// TwinCAT 3 PLC project TcCylinder
// Title: TcCylinder
// Company: TcNexa
// Author: ATI Software Engineering
// ProjectVersion: 2.2.0
// ProgramVersion: 3.1.4026.20
// libraries:
//   Tc2_Standard, * (Beckhoff Automation GmbH)
//   Tc2_System, * (Beckhoff Automation GmbH)
//   Tc3_Module, * (Beckhoff Automation GmbH)
//   TcDeviceBase, * (TcNexa)
//   TcProcess, * (TcNexa)
//   TcUnit, * (www.tcunit.org)
//   TcUtilities, * (TcNexa)
// project tree:
//   Cylinder/DUTs/ ST_CylinderConfig.TcDUT, ST_CylinderInfo.TcDUT
//   Cylinder/ITFs/ I_Cylinder.TcIO
//   Cylinder/POUs/ FB_Cylinder.TcPOU, FB_LiftCylinderBosch.TcPOU, FB_CylinderNexaHmi.TcPOU, FB_LiftCylinderNexaHmi_Bosch.TcPOU
//   / PlcTask.TcTTO
//   Tests/ FB_Cylinder_Test.TcPOU, PRG_TEST.TcPOU
//   Version/ Global_Version.TcGVL
// real-time tasks:
//   TASK PlcTask: cycle T#10ms, priority 20, ADS port 350

CONFIGURATION TcCylinder
    RESOURCE PLC ON TwinCAT3
        TASK PlcTask(INTERVAL := T#10ms, PRIORITY := 20);
        PROGRAM PRG_TEST WITH PlcTask : PRG_TEST;
    END_RESOURCE
END_CONFIGURATION

// ---- Cylinder/DUTs/ST_CylinderConfig.TcDUT
TYPE INTERNAL ST_CylinderConfig :
STRUCT
	delayTimeAfterReachedHP		: TIME;
	delayTimeAfterReachedWP		: TIME;
	movementTimeout				: TIME:= T#5S;
	monitorSensorsOverlap		: BOOL:= TRUE;
	sensorsOverlapTimeout		: TIME:= T#100MS;
END_STRUCT
END_TYPE

// ---- Cylinder/DUTs/ST_CylinderInfo.TcDUT
TYPE INTERNAL ST_CylinderInfo :
STRUCT
	sensorHP			: BOOL;
	sensorWP			: BOOL;
END_STRUCT
END_TYPE

// ---- Version/Global_Version.TcGVL
{attribute 'TcGenerated'}
{attribute 'no-analysis'}
{attribute 'linkalways'}
// This function has been automatically generated from the project information.
VAR_GLOBAL CONSTANT
	{attribute 'const_non_replaced'}
	stLibVersion_TcCylinder : ST_LibVersion := (iMajor := 2, iMinor := 2, iBuild := 0, iRevision := 0, nFlags := 0, sVersion := '2.2.0');
END_VAR

// ---- Cylinder/ITFs/I_Cylinder.TcIO
INTERFACE I_Cylinder

METHOD fill
VAR_INPUT
END_VAR
END_METHOD

PROPERTY PUBLIC inHP : BOOL
GET
END_GET
END_PROPERTY

PROPERTY PUBLIC inWP : BOOL
GET
END_GET
END_PROPERTY

METHOD PUBLIC moveToHP
VAR_INPUT
	Response		: REFERENCE TO TcNexa_Components_TcProcess.FB_MethodResponse;
END_VAR
END_METHOD

METHOD PUBLIC moveToWP
VAR_INPUT
	Response		: REFERENCE TO TcNexa_Components_TcProcess.FB_MethodResponse;
END_VAR
END_METHOD

METHOD PUBLIC off
VAR_INPUT
END_VAR
END_METHOD

END_INTERFACE

// ---- Tests/PRG_TEST.TcPOU
PROGRAM PRG_TEST
VAR
	_test : FB_Cylinder_Test;
END_VAR

TcUnit.RUN();

END_PROGRAM

// ---- Tests/FB_Cylinder_Test.TcPOU
FUNCTION_BLOCK FB_Cylinder_Test EXTENDS TcUnit.FB_TestSuite
VAR
END_VAR

testMoveToHP_BothSensorActive_Error();
testMoveToHP_MovementInterlocked_Error();
testMoveToHP_SensorNotReached_Timeout();
testMoveToHP_SensorNotUsed_Ok();
testMoveToHP_SensorReached_Ok();

METHOD PROTECTED testMoveToHP_BothSensorActive_Error
VAR_INST
	_testTimeout		: Tc2_Standard.TON;
	_Cylinder 			: FB_Cylinder	(name		:= 'Cylinder',
										tag			:= 'C1',
										sensorTagHP	:= 'B1',
										sensorTagWP	:= 'B2');
	_Response			: TcNexa_Components_TcProcess.FB_MethodResponse;
	_timerDelay			: Tc2_Standard.TON;
END_VAR
IF TcUnit.TEST_ORDERED(TestName:= 'TestMoveToHP_BothSensorActive_Error') THEN
	// Timeout if the movement is not executed right
	_testTimeout(IN:= TRUE, PT:= T#10S);
	_timerDelay(IN:= TRUE, PT:= T#1S);
	// Cylinder call
	_Cylinder.Config.delayTimeAfterReachedHP:= T#1S;	
	_Cylinder.FB_main();
	_Cylinder.moveToHP(Response:= _Response);
	TcUnit.WRITE_PROTECTED_BOOL(Ptr:= ADR(_Cylinder.sensorHP), Value:= _timerDelay.Q);
	TcUnit.WRITE_PROTECTED_BOOL(Ptr:= ADR(_Cylinder.sensorWP), Value:= TRUE);
	// Wait result
	IF _testTimeout.Q OR _Cylinder.inHP OR NOT _Response.busy THEN
		AssertFalse(
			Condition	:= _Cylinder.inHP,
			Message		:= 'inHP not FALSE');
		AssertFalse(
			Condition	:= _Cylinder.inWP,
			Message		:= 'inWP not FALSE');
		AssertFalse(
			Condition	:= _Response.busy,
			Message		:= 'busy not FALSE');
		AssertTrue(
			Condition	:= _Response.error,
			Message		:= 'error not TRUE');
			
		TcUnit.TEST_FINISHED();
	END_IF
END_IF
END_METHOD

METHOD PROTECTED testMoveToHP_MovementInterlocked_Error
VAR_INST
	_testTimeout		: Tc2_Standard.TON;
	_Cylinder 			: FB_Cylinder	(name		:= 'Cylinder',
										tag			:= 'C1',
										sensorTagHP	:= 'B1',
										sensorTagWP	:= 'B2');
	_Response			: TcNexa_Components_TcProcess.FB_MethodResponse;
	_timerDelay			: Tc2_Standard.TON;
END_VAR
IF TcUnit.TEST_ORDERED(TestName:= 'testMoveToHP_MovementInterlocked_Error') THEN
	// Timeout if the movement is not executed right
	_testTimeout(IN:= TRUE, PT:= T#10S);
	_timerDelay(IN:= TRUE, PT:= T#1S);
	// Cylinder call
	_Cylinder.addInterlockHP(condition:= TRUE, message:= '');
	_Cylinder.FB_main();
	_Cylinder.moveToHP(Response:= _Response);
	TcUnit.WRITE_PROTECTED_BOOL(Ptr:= ADR(_Cylinder.sensorHP), Value:= _timerDelay.Q);
	// Wait result
	IF _testTimeout.Q OR _Cylinder.inHP OR NOT _Response.busy THEN
		AssertFalse(
			Condition	:= _Cylinder.inHP,
			Message		:= 'inHP not FALSE');
		AssertFalse(
			Condition	:= _Cylinder.inWP,
			Message		:= 'inWP not FALSE');
		AssertFalse(
			Condition	:= _Response.busy,
			Message		:= 'busy not FALSE');
		AssertTrue(
			Condition	:= _Response.error,
			Message		:= 'error not TRUE');
			
		TcUnit.TEST_FINISHED();
	END_IF
END_IF
END_METHOD

METHOD PROTECTED testMoveToHP_SensorNotReached_Timeout
VAR_INST
	_testTimeout		: Tc2_Standard.TON;
	_Cylinder 			: FB_Cylinder	(name		:= 'Cylinder',
										tag			:= 'C1',
										sensorTagHP	:= 'B1',
										sensorTagWP	:= 'B2');
	_Response			: TcNexa_Components_TcProcess.FB_MethodResponse;
END_VAR
IF TcUnit.TEST_ORDERED(TestName:= 'TestMoveToHP_SensorNotReached_Timeout') THEN
	// Timeout if the movement is not executed right
	_testTimeout(IN:= TRUE, PT:= T#10S);
	// Cylinder call
	_Cylinder.FB_main();
	_Cylinder.moveToHP(Response:= _Response);
	// Wait result
	IF _testTimeout.Q OR _Cylinder.inHP OR NOT _Response.busy THEN
		AssertFalse(
			Condition	:= _Cylinder.inHP,
			Message		:= 'inHP not FALSE');
		AssertFalse(
			Condition	:= _Cylinder.inWP,
			Message		:= 'inWP not FALSE');
		AssertFalse(
			Condition	:= _Response.busy,
			Message		:= 'busy not FALSE');
		AssertTrue(
			Condition	:= _Response.error,
			Message		:= 'error not TRUE');
			
		TcUnit.TEST_FINISHED();
	END_IF
END_IF
END_METHOD

METHOD PROTECTED testMoveToHP_SensorNotUsed_Ok
VAR_INST
	_testTimeout		: Tc2_Standard.TON;
	_Cylinder 			: FB_Cylinder	(name		:= 'Cylinder',
										tag			:= 'C1',
										sensorTagHP	:= '',
										sensorTagWP	:= 'B2');
	_Response			: TcNexa_Components_TcProcess.FB_MethodResponse;
END_VAR
IF TcUnit.TEST_ORDERED(TestName:= 'testMoveToHP_SensorNotUsed_Ok') THEN
	// Timeout if the movement is not executed right
	_testTimeout(IN:= TRUE, PT:= T#10S);
	// Cylinder call
	_Cylinder.Config.delayTimeAfterReachedHP:= T#1S;
	_Cylinder.FB_main();
	_Cylinder.moveToHP(Response:= _Response);
	// Wait result
	IF _testTimeout.Q OR _Cylinder.inHP OR NOT _Response.busy THEN
		AssertTrue(
			Condition	:= _Cylinder.inHP,
			Message		:= 'inHP not TRUE');
		AssertFalse(
			Condition	:= _Cylinder.inWP,
			Message		:= 'inWP not FALSE');
		AssertFalse(
			Condition	:= _Response.busy,
			Message		:= 'busy not FALSE');
		AssertFalse(
			Condition	:= _Response.error,
			Message		:= 'error not FALSE');
			
		TcUnit.TEST_FINISHED();
	END_IF
END_IF
END_METHOD

METHOD PROTECTED testMoveToHP_SensorReached_Ok
VAR_INST
	_testTimeout		: Tc2_Standard.TON;
	_Cylinder 			: FB_Cylinder	(name		:= 'Cylinder',
										tag			:= 'C1',
										sensorTagHP	:= 'B1',
										sensorTagWP	:= 'B2');
	_Response			: TcNexa_Components_TcProcess.FB_MethodResponse;
	_timerDelay			: Tc2_Standard.TON;
END_VAR
IF TcUnit.TEST_ORDERED(TestName:= 'TestMoveToHP_SensorReached_Ok') THEN
	// Timeout if the movement is not executed right
	_testTimeout(IN:= TRUE, PT:= T#10S);
	_timerDelay(IN:= TRUE, PT:= T#1S);
	// Cylinder call
	_Cylinder.Config.delayTimeAfterReachedHP:= T#1S;	
	_Cylinder.FB_main();
	_Cylinder.moveToHP(Response:= _Response);
	TcUnit.WRITE_PROTECTED_BOOL(Ptr:= ADR(_Cylinder.sensorHP), Value:= _timerDelay.Q);
	// Wait result
	IF _testTimeout.Q OR _Cylinder.inHP OR NOT _Response.busy THEN
		AssertTrue(
			Condition	:= _Cylinder.inHP,
			Message		:= 'inHP not TRUE');
		AssertFalse(
			Condition	:= _Cylinder.inWP,
			Message		:= 'inWP not FALSE');
		AssertFalse(
			Condition	:= _Response.busy,
			Message		:= 'busy not FALSE');
		AssertFalse(
			Condition	:= _Response.error,
			Message		:= 'error not FALSE');
		AssertEquals_TIME(
			Expected	:= _timerDelay.ET + _Cylinder.Config.delayTimeAfterReachedHP + T#10MS,
			Actual		:= _testTimeout.ET,
			Message		:= 'delayTimeAfterReachedHP missmatch');
			
		TcUnit.TEST_FINISHED();
	END_IF
END_IF
END_METHOD

END_FUNCTION_BLOCK

// ---- Cylinder/POUs/FB_Cylinder.TcPOU
FUNCTION_BLOCK FB_Cylinder EXTENDS TcNexa_Devices_TcDeviceBase.FB_DeviceBase IMPLEMENTS I_Cylinder
VAR
(*----------------------------------------------------------------------------------------------*)
	sensorHP		AT %I*		: BOOL;
	sensorWP		AT %I*		: BOOL;
	valveHP			AT %Q*		: BOOL;
	valveWP			AT %Q*		: BOOL;
(*----------------------------------------------------------------------------------------------*)
	_Config						: ST_CylinderConfig;
	_Info						: ST_CylinderInfo;
	_inHP						: BOOL;
	_inWP						: BOOL;
	_newStateInterlockHP		: BOOL;
	_newStateInterlockMsgHP		: STRING(255);
	_interlockHP				: BOOL;
	_interlockMessageHP			: STRING(255);
	_newStateInterlockWP		: BOOL;
	_newStateInterlockMsgWP		: STRING(255);
	_interlockWP				: BOOL;
	_interlockMessageWP			: STRING(255);
	_sensorTagHP				: STRING;
	_sensorTagWP				: STRING;
	_notUsedSensorHP			: BOOL;
	_notUsedSensorWP			: BOOL;
	_timerTimeout				: Tc2_Standard.TON;
	_timerSensorsOverlap		: Tc2_Standard.TON;
	_timerInHP					: Tc2_Standard.TON;
	_timerInWP					: Tc2_Standard.TON;
(*----------------------------------------------------------------------------------------------*)
END_VAR

METHOD INTERNAL _getErrorMsgPositionNotReached : STRING(255)
VAR_INPUT
	sensor		: STRING;
END_VAR
_getErrorMsgPositionNotReached:= 'Position not reached';
IF (sensor <> '') THEN
	_getErrorMsgPositionNotReached:= Tc2_Standard.CONCAT(STR1:= _getErrorMsgPositionNotReached, STR2:= ' (');
	_getErrorMsgPositionNotReached:= Tc2_Standard.CONCAT(STR1:= _getErrorMsgPositionNotReached, STR2:= sensor);
	_getErrorMsgPositionNotReached:= Tc2_Standard.CONCAT(STR1:= _getErrorMsgPositionNotReached, STR2:= ')');
END_IF
END_METHOD

METHOD INTERNAL _getMsgInterlocked : STRING(255)
VAR_INPUT
END_VAR
_getMsgInterlocked:= Tc2_Standard.CONCAT(STR1:= _nameTag, STR2:= ' interlocked during ');
_getMsgInterlocked:= Tc2_Standard.CONCAT(STR1:= _getMsgInterlocked, STR2:= _calledMethod);
END_METHOD

METHOD INTERNAL _handleInterlocks
VAR_INPUT
END_VAR
(*----------------------------------------------------------------------------------------------*)
_interlockHP:= _newStateInterlockHP;
_interlockMessageHP:= _newStateInterlockMsgHP;
_newStateInterlockHP:= FALSE;
_newStateInterlockMsgHP:= '';
(*----------------------------------------------------------------------------------------------*)
_interlockWP:= _newStateInterlockWP;
_interlockMessageWP:= _newStateInterlockMsgWP;
_newStateInterlockWP:= FALSE;
_newStateInterlockMsgWP:= '';
(*----------------------------------------------------------------------------------------------*)
END_METHOD

METHOD INTERNAL _handlePositionStatus
VAR_INPUT
END_VAR
(*----------------------------------------------------------------------------------------------*)
_timerInHP(
	IN	:= valveHP AND (_notUsedSensorHP OR sensorHP) AND (NOT sensorWP OR NOT _Config.monitorSensorsOverlap),
	PT	:= _Config.delayTimeAfterReachedHP,
	Q	=> _inHP);
(*----------------------------------------------------------------------------------------------*)
_timerInWP(
	IN	:= valveWP AND (_notUsedSensorWP OR sensorWP) AND (NOT sensorHP OR NOT _Config.monitorSensorsOverlap),
	PT	:= _Config.delayTimeAfterReachedWP,
	Q	=> _inWP);
(*----------------------------------------------------------------------------------------------*)
_timerTimeout(
	IN:= (_calledMethod <> ''),
	PT:= _Config.movementTimeout);
(*----------------------------------------------------------------------------------------------*)
_timerSensorsOverlap(
	IN:= _Config.monitorSensorsOverlap AND sensorHP AND sensorWP,
	PT:= _Config.sensorsOverlapTimeout);
(*----------------------------------------------------------------------------------------------*)
END_METHOD

METHOD PROTECTED _methodHeader : ST_MethodState
VAR_INPUT
	methodName		: Tc2_System.T_MaxString;
END_VAR
IF (_calledMethod = '') THEN
	_timerTimeout(IN:= FALSE);
	_timerSensorsOverlap(IN:= FALSE);
	_calledMethod:= methodName;
	_Step.init();
	_methodTimeout(IN:= FALSE);
	_methodHeader.init:= TRUE;
	_methodHeader.execute:= TRUE;
	_executeMethod:= TRUE;
	_InternalResponse.setBusy(message:= methodName);
ELSIF (_calledMethod = methodName) THEN
	_executeMethod:= TRUE;
	_tmpText:= _getBusyMessage(message:= 'in progress');
	_InternalResponse.setBusy(message:= _tmpText);
	_methodHeader.execute:= TRUE;
ELSE
	_tmpText:= _getBusyMessage(message:= 'in progress');
	_InternalResponse.setBusy(message:= _tmpText);
END_IF
END_METHOD

METHOD PROTECTED _onInit
VAR_INST
	_isInit				: BOOL;
END_VAR
(*----------------------------------------------------------------------------------------------*)
IF _isInit THEN RETURN; END_IF
(*----------------------------------------------------------------------------------------------*)
IF (_sensorTagHP = '') THEN
	_notUsedSensorHP:= TRUE;
END_IF
(*----------------------------------------------------------------------------------------------*)
IF (_sensorTagWP = '') THEN
	_notUsedSensorWP:= TRUE;
END_IF
(*----------------------------------------------------------------------------------------------*)
_isInit:= TRUE;
(*----------------------------------------------------------------------------------------------*)
END_METHOD

METHOD INTERNAL _updateInfo
VAR_INPUT
END_VAR
_Info.sensorHP:= sensorHP;
_Info.sensorWP:= sensorWP;
END_METHOD

METHOD addInterlockHP
VAR_INPUT
	condition		: BOOL;
	message			: STRING(255);
END_VAR
IF condition THEN
	_newStateInterlockHP:= TRUE;
	_newStateInterlockMsgHP:= message;
END_IF
END_METHOD

METHOD addInterlockWP
VAR_INPUT
	condition		: BOOL;
	message			: STRING(255);
END_VAR
IF condition THEN
	_newStateInterlockWP:= TRUE;
	_newStateInterlockMsgWP:= message;
END_IF
END_METHOD

PROPERTY Config : REFERENCE TO ST_CylinderConfig
GET
Config REF= _Config;
END_GET
END_PROPERTY

METHOD FB_init : BOOL
VAR_INPUT
	bInitRetains 	: BOOL; 	// if TRUE, the retain variables are initialized (warm start / cold start)
	bInCopyCode 	: BOOL;  	// if TRUE, the instance afterwards gets moved into the copy code (online change)
	name			: STRING;	// identifier for HMI display and logging, example Clipping cylinder
	tag				: STRING;	// el. schematic tag for device, example C1, 10MM1, Z1, etc.
	sensorTagHP		: STRING;	// el. schematic tag for home position sensor input, leave empty '' if no HP sensor attached
	sensorTagWP		: STRING;	// el. schematic tag for work position sensor input, leave empty '' if no WP sensor attached
END_VAR
THIS^._sensorTagHP:= sensorTagHP;
THIS^._sensorTagWP:= sensorTagWP;
END_METHOD

METHOD PUBLIC FB_main
VAR_INPUT
END_VAR
SUPER^.FB_main();

_onInit();
_handleInterlocks();
_handlePositionStatus();
_updateInfo();
END_METHOD

METHOD fill
VAR_INPUT
END_VAR
valveHP:= TRUE;
valveWP:= TRUE;
END_METHOD

PROPERTY Info : REFERENCE TO ST_CylinderInfo
GET
Info REF= _Info;
END_GET
END_PROPERTY

PROPERTY PUBLIC inHP : BOOL
GET
inHP:= _inHP;
END_GET
END_PROPERTY

PROPERTY PUBLIC inWP : BOOL
GET
inWP:= _inWP;
END_GET
END_PROPERTY

METHOD PUBLIC moveToHP
VAR_INPUT
	Response		: REFERENCE TO TcNexa_Components_TcProcess.FB_MethodResponse;
END_VAR
_methodState:= _methodHeader(methodName:= 'move to HP');

IF _methodState.execute THEN
	IF NOT _interlockHP THEN
		valveHP:= TRUE;
		valveWP:= FALSE;		
		(* Error - both sensors active *)
		IF _timerSensorsOverlap.Q THEN
			_InternalResponse.setFail(message:= _getErrorMessage(), description:= 'Both sensors active');
		(* Error movement - end position not reached *)		
		ELSIF _timerTimeout.Q THEN
			_InternalResponse.setFail(message:= _getErrorMessage(), description:= _getErrorMsgPositionNotReached(_sensorTagHP));
		(* Succes - end position reached *)
		ELSIF _timerInHP.Q THEN
			_InternalResponse.setPass();
		END_IF
	ELSE
		_InternalResponse.setFail(message:= _getMsgInterlocked(), description:= _interlockMessageHP);
	END_IF
END_IF

_methodFooter(Response:= Response);
END_METHOD

METHOD PUBLIC moveToWP
VAR_INPUT
	Response		: REFERENCE TO TcNexa_Components_TcProcess.FB_MethodResponse;
END_VAR
_methodState:= _methodHeader(methodName:= 'move to WP');

IF _methodState.execute THEN
	IF NOT _interlockWP THEN
		valveHP:= FALSE;
		valveWP:= TRUE;		
	
		(* Error - both sensors active *)
		IF _timerSensorsOverlap.Q THEN
			_InternalResponse.setFail(message:= _getErrorMessage(), description:= 'Both sensors active');
		(* Error movement - end position not reached *)		
		ELSIF _timerTimeout.Q THEN
			_InternalResponse.setFail(message:= _getErrorMessage(), description:= _getErrorMsgPositionNotReached(_sensorTagWP));
		(* Succes - end position reached *)
		ELSIF _timerInWP.Q THEN
			_InternalResponse.setPass();
		END_IF	
	ELSE
		_InternalResponse.setFail(message:= _getMsgInterlocked(), description:= _interlockMessageWP);
	END_IF
END_IF

_methodFooter(Response:= Response);
END_METHOD

METHOD PUBLIC off
VAR_INPUT
END_VAR
valveHP:= FALSE;
valveWP:= FALSE;
END_METHOD

END_FUNCTION_BLOCK

// ---- Cylinder/POUs/FB_LiftCylinderBosch.TcPOU
FUNCTION_BLOCK FB_LiftCylinderBosch EXTENDS FB_Cylinder
VAR
(*----------------------------------------------------------------------------------------------*)
	sensorMID		AT %I*		: BOOL;
(*----------------------------------------------------------------------------------------------*)
	_inMID						: BOOL;
	_newStateInterlockMID		: BOOL;
	_newStateInterlockMsgMID	: STRING(255);
	_interlockMID				: BOOL;
	_interlockMessageMID		: STRING(255);
	_sensorTagMID				: STRING;
	_notUsedSensorMID			: BOOL;
	_delayTimeAfterReachedMID	: TIME;
	_timerInMID					: Tc2_Standard.TON;	
(*----------------------------------------------------------------------------------------------*)
END_VAR

METHOD INTERNAL _handleInterlocks
VAR_INPUT
END_VAR
(*----------------------------------------------------------------------------------------------*)
_interlockHP:= _newStateInterlockHP;
_interlockMessageHP:= _newStateInterlockMsgHP;
_newStateInterlockHP:= FALSE;
_newStateInterlockMsgHP:= '';
(*----------------------------------------------------------------------------------------------*)
_interlockMID:= _newStateInterlockMID;
_interlockMessageMID:= _newStateInterlockMsgMID;
_newStateInterlockMID:= FALSE;
_newStateInterlockMsgMID:= '';
(*----------------------------------------------------------------------------------------------*)
_interlockWP:= _newStateInterlockWP;
_interlockMessageWP:= _newStateInterlockMsgWP;
_newStateInterlockWP:= FALSE;
_newStateInterlockMsgWP:= '';
(*----------------------------------------------------------------------------------------------*)
END_METHOD

METHOD INTERNAL _handlePositionStatus
VAR_INPUT
END_VAR
(*----------------------------------------------------------------------------------------------*)
_timerInHP(
	IN	:= valveHP AND (_notUsedSensorHP OR sensorHP) AND (NOT sensorWP OR NOT _Config.monitorSensorsOverlap),
	PT	:= _Config.delayTimeAfterReachedHP,
	Q	=> _inHP);
(*----------------------------------------------------------------------------------------------*)
_timerInMID(
	IN	:= NOT valveHP AND NOT valveWP AND (_notUsedSensorMID OR sensorMID) AND (NOT sensorHP OR NOT _Config.monitorSensorsOverlap) AND (NOT sensorWP OR NOT _Config.monitorSensorsOverlap),
	PT	:= _delayTimeAfterReachedMID,
	Q	=> _inMID);
(*----------------------------------------------------------------------------------------------*)
_timerInWP(
	IN	:= valveWP AND (_notUsedSensorWP OR sensorWP) AND (NOT sensorHP OR NOT _Config.monitorSensorsOverlap),
	PT	:= _Config.delayTimeAfterReachedWP,
	Q	=> _inWP);
(*----------------------------------------------------------------------------------------------*)
_timerTimeout(
	IN:= (_calledMethod <> ''),
	PT:= _Config.movementTimeout);
(*----------------------------------------------------------------------------------------------*)
_timerSensorsOverlap(
	IN:= _Config.monitorSensorsOverlap AND sensorHP AND sensorWP,
	PT:= _Config.sensorsOverlapTimeout);
(*----------------------------------------------------------------------------------------------*)
END_METHOD

METHOD PROTECTED _onInit
VAR_INST
	_isInit				: BOOL;
END_VAR
(*----------------------------------------------------------------------------------------------*)
IF _isInit THEN RETURN; END_IF
(*----------------------------------------------------------------------------------------------*)
IF (_sensorTagHP = '') THEN
	_notUsedSensorHP:= TRUE;
END_IF
(*----------------------------------------------------------------------------------------------*)
IF (_sensorTagMID = '') THEN
	_notUsedSensorMID:= TRUE;
END_IF
(*----------------------------------------------------------------------------------------------*)
IF (_sensorTagWP = '') THEN
	_notUsedSensorWP:= TRUE;
END_IF
(*----------------------------------------------------------------------------------------------*)
_isInit:= TRUE;
(*----------------------------------------------------------------------------------------------*)
END_METHOD

METHOD addInterlockMID
VAR_INPUT
	condition		: BOOL;
	message			: STRING(255);
END_VAR
IF condition THEN
	_newStateInterlockMID:= TRUE;
	_newStateInterlockMsgMID:= message;
END_IF
END_METHOD

PROPERTY delayTimeAfterReachedMID : TIME
GET
delayTimeAfterReachedMID:= _delayTimeAfterReachedMID;
END_GET
SET
_delayTimeAfterReachedMID:= delayTimeAfterReachedMID;
END_SET
END_PROPERTY

METHOD FB_init : BOOL
VAR_INPUT
	bInitRetains 	: BOOL; 	// if TRUE, the retain variables are initialized (warm start / cold start)
	bInCopyCode 	: BOOL;  	// if TRUE, the instance afterwards gets moved into the copy code (online change)
	name			: STRING;	// identifier for HMI display and logging, example Clipping cylinder
	tag				: STRING;	// el. schematic tag for device, example C1, 10MM1, Z1, etc.
	sensorTagHP		: STRING;	// el. schematic tag for home position sensor input, leave empty '' if no HP sensor attached
	sensorTagWP		: STRING;	// el. schematic tag for work position sensor input, leave empty '' if no WP sensor attached
	sensorTagMID	: STRING;	// el. schematic tag for mid position sensor input, leave empty '' if no MID sensor attached
END_VAR
THIS^._sensorTagMID:= sensorTagMID;
END_METHOD

PROPERTY PUBLIC inMID : BOOL
GET
inMID:= _inMID;
END_GET
END_PROPERTY

METHOD PUBLIC moveToMID
VAR_INPUT
	Response		: REFERENCE TO TcNexa_Components_TcProcess.FB_MethodResponse;
END_VAR
_methodState:= _methodHeader(methodName:= 'move to MID');

IF _methodState.execute THEN
	IF NOT _interlockMID THEN
		valveHP:= FALSE;
		valveWP:= FALSE;		
		(* Error - all sensors active *)
		IF _timerSensorsOverlap.Q THEN
			_InternalResponse.setFail(message:= _getErrorMessage(), description:= 'All sensors active');
		(* Error movement - end position not reached *)		
		ELSIF _timerTimeout.Q THEN
			_InternalResponse.setFail(message:= _getErrorMessage(), description:= _getErrorMsgPositionNotReached(_sensorTagMID));
		(* Succes - end position reached *)
		ELSIF _timerInMID.Q THEN
			_InternalResponse.setPass();
		END_IF	
	ELSE
		_InternalResponse.setFail(message:= _getMsgInterlocked(), description:= _interlockMessageMID);
	END_IF
END_IF

_methodFooter(Response:= Response);
END_METHOD

END_FUNCTION_BLOCK

// ---- Cylinder/POUs/FB_CylinderNexaHmi.TcPOU
FUNCTION_BLOCK FB_CylinderNexaHmi EXTENDS FB_Cylinder
VAR
	(* Hmi *)       			
	_Hmi						: TcNexa_Devices_TcDeviceBase.FB_DeviceNexaHmi(deviceType:= 'cylinders');
	_onHmiConnection			: Tc2_Standard.R_TRIG;
	_isHmiConnected				: BOOL;
	_commandNameHP				: STRING;
	_commandNameWP				: STRING;
	_manualMode					: BOOL;
	_onResponseError			: Tc2_Standard.R_TRIG;
	_onResponsePass				: Tc2_Standard.R_TRIG;
	_interlockHPforOtherDevices	: STRING;
	_interlockWPforOtherDevices	: STRING;
	(* Control VAR *)
	_lastNotUsedSensorHP		: BOOL;
	_lastSensorHP				: BOOL;
	_lastNotUsedSensorWP		: BOOL;
	_lastSensorWP				: BOOL;
	_message					: STRING(255);
	_lastMessage				: STRING(255);
	(* Buttons *)
	_ButtonHP					: TcNexa_Devices_TcDeviceBase.FB_DeviceButtonNexaHmi(
									Hmi			:= _Hmi, 
									topic		:= 'general/buttons/HP/');
	_ButtonWP					: TcNexa_Devices_TcDeviceBase.FB_DeviceButtonNexaHmi(
									Hmi			:= _Hmi, 
									topic		:= 'general/buttons/WP/');
	(* Commands *)
	_requestHP					: BOOL;
	_requestWP					: BOOL;
END_VAR

METHOD PROTECTED _handleButtons
VAR_INPUT
END_VAR
(*----------------------------------------------------------------------------------------------*)
_ButtonHP.enabled:= NOT _interlockHP AND _manualMode;
_ButtonHP.focused:= valveHP;
_ButtonHP.name:= _commandNameHP;
_ButtonHP.FB_main();
(*----------------------------------------------------------------------------------------------*)
_ButtonWP.enabled:= NOT _interlockWP AND _manualMode;
_ButtonWP.focused:= valveWP;
_ButtonWP.name:= _commandNameWP;
_ButtonWP.FB_main();
(*----------------------------------------------------------------------------------------------*)
IF NOT _manualMode THEN RETURN; END_IF
IF _ButtonHP.onTap THEN	_requestHP:= TRUE; END_IF
IF _ButtonWP.onTap THEN	_requestWP:= TRUE; END_IF
(*----------------------------------------------------------------------------------------------*)
END_METHOD

METHOD PROTECTED _handleManual
VAR_INPUT
END_VAR
IF NOT _manualMode THEN
	_requestHP:= FALSE;
	_requestWP:= FALSE;
	_message:= 'Movement blocked: Not in manual mode';
ELSIF _interlockHP AND NOT _inHP THEN
	_message:= Tc2_Standard.CONCAT(STR1:= _commandNameHP, ' blocked: ');
	_message:= Tc2_Standard.CONCAT(STR1:= _message, _interlockMessageHP);
ELSIF _interlockWP AND NOT _inWP THEN
	_message:= Tc2_Standard.CONCAT(STR1:= _commandNameWP, ' blocked: ');
	_message:= Tc2_Standard.CONCAT(STR1:= _message, _interlockMessageWP);
ELSE
	_message:= '';
	(* HP *)
	IF _requestHP THEN
		moveToHP(Response:= _InternalResponse);
		_requestHP:= FALSE;
	END_IF
	(* HP *)
	IF _requestWP THEN
		moveToWP(Response:= _InternalResponse);
		_requestWP:= FALSE;
	END_IF
END_IF
END_METHOD

METHOD PROTECTED _onConnection
VAR_INPUT
END_VAR
IF NOT _onHmiConnection.Q THEN RETURN; END_IF

(* Publish *)
_Hmi.publish(
	topic	:= 'general/sensorTagHP',
	payload	:= _sensorTagHP);
_Hmi.publish(
	topic	:= 'general/sensorTagWP',
	payload	:= _sensorTagWP);
END_METHOD

METHOD PROTECTED _publishTopics
VAR_INPUT
END_VAR
IF NOT _isHmiConnected THEN RETURN; END_IF
(*----------------------------------------------------------------------------------------------*)
IF (_lastNotUsedSensorHP <> _notUsedSensorHP) OR _onHmiConnection.Q THEN
	_lastNotUsedSensorHP:= _notUsedSensorHP;
	_Hmi.publish(
		topic	:= 'general/notUsedSensorHP',
		payload	:= BOOL_TO_STRING(_notUsedSensorHP));
END_IF
(*----------------------------------------------------------------------------------------------*)
IF (_lastSensorHP <> sensorHP) OR _onHmiConnection.Q THEN
	_lastSensorHP:= sensorHP;
	_Hmi.publish(
		topic	:= 'general/sensorHP',
		payload	:= BOOL_TO_STRING(sensorHP));
END_IF
(*----------------------------------------------------------------------------------------------*)
IF (_lastNotUsedSensorWP <> _notUsedSensorWP) OR _onHmiConnection.Q THEN
	_lastNotUsedSensorWP:= _notUsedSensorWP;
	_Hmi.publish(
		topic	:= 'general/notUsedSensorWP',
		payload	:= BOOL_TO_STRING(_notUsedSensorWP));
END_IF
(*----------------------------------------------------------------------------------------------*)
IF (_lastSensorWP <> sensorWP) OR _onHmiConnection.Q THEN
	_lastSensorWP:= sensorWP;
	_Hmi.publish(
		topic	:= 'general/sensorWP',
		payload	:= BOOL_TO_STRING(sensorWP));
END_IF
(*----------------------------------------------------------------------------------------------*)
IF (_message <> _lastMessage) OR _onHmiConnection.Q THEN
	_lastMessage:= _message;
	_Hmi.publish(
		topic	:= 'general/message',
		payload	:= _message);
END_IF
(*----------------------------------------------------------------------------------------------*)
END_METHOD

METHOD FB_init : BOOL
VAR_INPUT
	bInitRetains 	: BOOL; // if TRUE, the retain variables are initialized (warm start / cold start)
	bInCopyCode 	: BOOL;  // if TRUE, the instance afterwards gets moved into the copy code (online change)
	name			: STRING;
	tag				: STRING;
	sensorTagHP		: STRING;
	sensorTagWP		: STRING;
	commandNameHP	: STRING;
	commandNameWP	: STRING;
	cellTag			: STRING;
	stationTag		: STRING;
END_VAR
THIS^._commandNameHP:= commandNameHP;
THIS^._commandNameWP:= commandNameWP;

THIS^._Hmi.cellTag:= cellTag;
THIS^._Hmi.stationTag:= stationTag;
THIS^._Hmi.deviceTag:= tag;
THIS^._Hmi.deviceName:= name;

_interlockHPforOtherDevices:= Tc2_Standard.CONCAT(STR1:= _nameTag, STR2:= ' not in ');
_interlockHPforOtherDevices:= Tc2_Standard.CONCAT(STR1:= _interlockHPforOtherDevices, STR2:= _commandNameHP);
_interlockHPforOtherDevices:= Tc2_Standard.CONCAT(STR1:= _interlockHPforOtherDevices, STR2:= ' position');
_interlockWPforOtherDevices:= Tc2_Standard.CONCAT(STR1:= _nameTag, STR2:= ' not in ');
_interlockWPforOtherDevices:= Tc2_Standard.CONCAT(STR1:= _interlockWPforOtherDevices, STR2:= _commandNameWP);
_interlockWPforOtherDevices:= Tc2_Standard.CONCAT(STR1:= _interlockWPforOtherDevices, STR2:= ' position');
END_METHOD

METHOD PUBLIC FB_main
VAR_INPUT
END_VAR
SUPER^.FB_main();
_Hmi.FB_main();
_isHmiConnected:= _Hmi.isConnected;
_onHmiConnection(CLK:= _isHmiConnected);

_onConnection();
_publishTopics();
_handleButtons();
_handleManual();
END_METHOD

PROPERTY PUBLIC hostName : Tc2_System.T_MaxString
GET
hostName:= _Hmi.hostName;
END_GET
SET
_Hmi.hostName:= hostName;
END_SET
END_PROPERTY

PROPERTY PUBLIC hostPort : UINT
GET
hostPort:= _Hmi.hostPort;
END_GET
SET
_Hmi.hostPort:= hostPort;
END_SET
END_PROPERTY

PROPERTY interlockMessageHP : STRING(255)
GET
interlockMessageHP:= _interlockHPforOtherDevices;
END_GET
END_PROPERTY

PROPERTY interlockMessageWP : STRING(255)
GET
interlockMessageWP:= _interlockWPforOtherDevices;
END_GET
END_PROPERTY

PROPERTY manualMode : BOOL
GET
manualMode:= _manualMode;
END_GET
SET
_manualMode:= manualMode;
END_SET
END_PROPERTY

END_FUNCTION_BLOCK

// ---- Cylinder/POUs/FB_LiftCylinderNexaHmi_Bosch.TcPOU
FUNCTION_BLOCK FB_LiftCylinderNexaHmi_Bosch EXTENDS FB_LiftCylinderBosch
VAR
(*----------------------------------------------------------------------------------------------*)
	_Hmi						: TcNexa_Devices_TcDeviceBase.FB_DeviceNexaHmi(deviceType:= 'cylinders3pos');
	_onHmiConnection			: Tc2_Standard.R_TRIG;
	_isHmiConnected				: BOOL;
	_commandNameHP				: STRING;
	_commandNameMID				: STRING;
	_commandNameWP				: STRING;
	_manualMode					: BOOL;
	_onResponseError			: Tc2_Standard.R_TRIG;
	_onResponsePass				: Tc2_Standard.R_TRIG;
	_interlockHPforOtherDevices	: STRING;
	_interlockMIDforOtherDevices: STRING;
	_interlockWPforOtherDevices	: STRING;
	(* Control VAR *)
	_lastNotUsedSensorHP		: BOOL;
	_lastSensorHP				: BOOL;
	_lastNotUsedSensorMID		: BOOL;
	_lastSensorMID				: BOOL;
	_lastNotUsedSensorWP		: BOOL;
	_lastSensorWP				: BOOL;
	_message					: STRING(255);
	_lastMessage				: STRING(255);
(*----------------------------------------------------------------------------------------------*)
	_ButtonHP					: TcNexa_Devices_TcDeviceBase.FB_DeviceButtonNexaHmi(
									Hmi			:= _Hmi, 
									topic		:= 'general/buttons/1/');
	_ButtonMID					: TcNexa_Devices_TcDeviceBase.FB_DeviceButtonNexaHmi(
									Hmi			:= _Hmi, 
									topic		:= 'general/buttons/2/');
	_ButtonWP					: TcNexa_Devices_TcDeviceBase.FB_DeviceButtonNexaHmi(
									Hmi			:= _Hmi, 
									topic		:= 'general/buttons/3/');
(*----------------------------------------------------------------------------------------------*)
	_requestHP					: BOOL;
	_requestMID					: BOOL;
	_requestWP					: BOOL;
(*----------------------------------------------------------------------------------------------*)
END_VAR

METHOD PROTECTED _handleButtons
VAR_INPUT
END_VAR
(*----------------------------------------------------------------------------------------------*)
_ButtonHP.enabled:= NOT _interlockHP AND _manualMode;
_ButtonHP.focused:= valveHP;
_ButtonHP.name:= _commandNameHP;
_ButtonHP.FB_main();
(*----------------------------------------------------------------------------------------------*)
_ButtonMID.enabled:= NOT _interlockMID AND _manualMode;
_ButtonMID.focused:= NOT valveHP AND NOT valveWP;
_ButtonMID.name:= _commandNameMID;
_ButtonMID.FB_main();
(*----------------------------------------------------------------------------------------------*)
_ButtonWP.enabled:= NOT _interlockWP AND _manualMode;
_ButtonWP.focused:= valveWP;
_ButtonWP.name:= _commandNameWP;
_ButtonWP.FB_main();
(*----------------------------------------------------------------------------------------------*)
IF NOT _manualMode THEN RETURN; END_IF
IF _ButtonHP.onTap THEN	_requestHP:= TRUE; END_IF
IF _ButtonMID.onTap THEN _requestMID:= TRUE; END_IF
IF _ButtonWP.onTap THEN	_requestWP:= TRUE; END_IF
(*----------------------------------------------------------------------------------------------*)
END_METHOD

METHOD PROTECTED _handleManual
VAR_INPUT
END_VAR
IF NOT _manualMode THEN
	_requestHP:= FALSE;
	_requestMID:= FALSE;
	_requestWP:= FALSE;
	_message:= 'Movement blocked: Not in manual mode';
ELSIF _interlockHP AND NOT _inHP THEN
	_message:= Tc2_Standard.CONCAT(STR1:= _commandNameHP, ' blocked: ');
	_message:= Tc2_Standard.CONCAT(STR1:= _message, _interlockMessageHP);
ELSIF _interlockMID AND NOT _inMID THEN
	_message:= Tc2_Standard.CONCAT(STR1:= _commandNameHP, ' blocked: ');
	_message:= Tc2_Standard.CONCAT(STR1:= _message, _interlockMessageMID);
ELSIF _interlockWP AND NOT _inWP THEN
	_message:= Tc2_Standard.CONCAT(STR1:= _commandNameWP, ' blocked: ');
	_message:= Tc2_Standard.CONCAT(STR1:= _message, _interlockMessageWP);
ELSE
	_message:= '';
	(* HP *)
	IF _requestHP THEN
		moveToHP(Response:= _InternalResponse);
		_requestHP:= FALSE;
	END_IF
	(* MID *)
	IF _requestMID THEN
		moveToMID(Response:= _InternalResponse);
		_requestMID:= FALSE;
	END_IF
	(* WP *)
	IF _requestWP THEN
		moveToWP(Response:= _InternalResponse);
		_requestWP:= FALSE;
	END_IF
END_IF
END_METHOD

METHOD PROTECTED _onConnection
VAR_INPUT
END_VAR
IF NOT _onHmiConnection.Q THEN RETURN; END_IF

(* Publish *)
_Hmi.publish(
	topic	:= 'general/sensorTag1',
	payload	:= _sensorTagHP);
_Hmi.publish(
	topic	:= 'general/sensorTag2',
	payload	:= _sensorTagMID);
_Hmi.publish(
	topic	:= 'general/sensorTag3',
	payload	:= _sensorTagWP);
END_METHOD

METHOD PROTECTED _publishTopics
VAR_INPUT
END_VAR
IF NOT _isHmiConnected THEN RETURN; END_IF
(*----------------------------------------------------------------------------------------------*)
IF (_lastNotUsedSensorHP <> _notUsedSensorHP) OR _onHmiConnection.Q THEN
	_lastNotUsedSensorHP:= _notUsedSensorHP;
	_Hmi.publish(
		topic	:= 'general/notUsedSensorHP',
		payload	:= BOOL_TO_STRING(_notUsedSensorHP));
END_IF
(*----------------------------------------------------------------------------------------------*)
IF (_lastSensorHP <> sensorHP) OR _onHmiConnection.Q THEN
	_lastSensorHP:= sensorHP;
	_Hmi.publish(
		topic	:= 'general/sensorHP',
		payload	:= BOOL_TO_STRING(sensorHP));
END_IF
(*----------------------------------------------------------------------------------------------*)
IF (_lastNotUsedSensorMID <> _notUsedSensorMID) OR _onHmiConnection.Q THEN
	_lastNotUsedSensorMID:= _notUsedSensorMID;
	_Hmi.publish(
		topic	:= 'general/notUsedSensorMID',
		payload	:= BOOL_TO_STRING(_notUsedSensorMID));
END_IF
(*----------------------------------------------------------------------------------------------*)
IF (_lastSensorMID <> sensorMID) OR _onHmiConnection.Q THEN
	_lastSensorMID:= sensorMID;
	_Hmi.publish(
		topic	:= 'general/sensorMID',
		payload	:= BOOL_TO_STRING(sensorMID));
END_IF
(*----------------------------------------------------------------------------------------------*)
IF (_lastNotUsedSensorWP <> _notUsedSensorWP) OR _onHmiConnection.Q THEN
	_lastNotUsedSensorWP:= _notUsedSensorWP;
	_Hmi.publish(
		topic	:= 'general/notUsedSensorWP',
		payload	:= BOOL_TO_STRING(_notUsedSensorWP));
END_IF
(*----------------------------------------------------------------------------------------------*)
IF (_lastSensorWP <> sensorWP) OR _onHmiConnection.Q THEN
	_lastSensorWP:= sensorWP;
	_Hmi.publish(
		topic	:= 'general/sensorWP',
		payload	:= BOOL_TO_STRING(sensorWP));
END_IF
(*----------------------------------------------------------------------------------------------*)
IF (_message <> _lastMessage) OR _onHmiConnection.Q THEN
	_lastMessage:= _message;
	_Hmi.publish(
		topic	:= 'general/message',
		payload	:= _message);
END_IF
(*----------------------------------------------------------------------------------------------*)
END_METHOD

METHOD FB_init : BOOL
VAR_INPUT
	bInitRetains 	: BOOL; // if TRUE, the retain variables are initialized (warm start / cold start)
	bInCopyCode 	: BOOL;  // if TRUE, the instance afterwards gets moved into the copy code (online change)
	name			: STRING;
	tag				: STRING;
	sensorTagHP		: STRING;
	sensorTagWP		: STRING;
	sensorTagMID	: STRING;
	commandNameHP	: STRING;
	commandNameMID	: STRING;
	commandNameWP	: STRING;
	cellTag			: STRING;
	stationTag		: STRING;
END_VAR
THIS^._commandNameHP:= commandNameHP;
THIS^._commandNameMID:= commandNameMID;
THIS^._commandNameWP:= commandNameWP;

THIS^._Hmi.cellTag:= cellTag;
THIS^._Hmi.stationTag:= stationTag;
THIS^._Hmi.deviceTag:= tag;
THIS^._Hmi.deviceName:= name;

_interlockHPforOtherDevices:= Tc2_Standard.CONCAT(STR1:= _nameTag, STR2:= ' not in ');
_interlockHPforOtherDevices:= Tc2_Standard.CONCAT(STR1:= _interlockHPforOtherDevices, STR2:= _commandNameHP);
_interlockHPforOtherDevices:= Tc2_Standard.CONCAT(STR1:= _interlockHPforOtherDevices, STR2:= ' position');
_interlockWPforOtherDevices:= Tc2_Standard.CONCAT(STR1:= _nameTag, STR2:= ' not in ');
_interlockWPforOtherDevices:= Tc2_Standard.CONCAT(STR1:= _interlockWPforOtherDevices, STR2:= _commandNameWP);
_interlockWPforOtherDevices:= Tc2_Standard.CONCAT(STR1:= _interlockWPforOtherDevices, STR2:= ' position');
END_METHOD

METHOD PUBLIC FB_main
VAR_INPUT
END_VAR
SUPER^.FB_main();
_Hmi.FB_main();
_isHmiConnected:= _Hmi.isConnected;
_onHmiConnection(CLK:= _isHmiConnected);

_onConnection();
_publishTopics();
_handleButtons();
_handleManual();
END_METHOD

PROPERTY PUBLIC hostName : Tc2_System.T_MaxString
GET
hostName:= _Hmi.hostName;
END_GET
SET
_Hmi.hostName:= hostName;
END_SET
END_PROPERTY

PROPERTY PUBLIC hostPort : UINT
GET
hostPort:= _Hmi.hostPort;
END_GET
SET
_Hmi.hostPort:= hostPort;
END_SET
END_PROPERTY

PROPERTY interlockMessageHP : STRING(255)
GET
interlockMessageHP:= _interlockHPforOtherDevices;
END_GET
END_PROPERTY

PROPERTY interlockMessageMID : STRING(255)
GET
interlockMessageMID:= _interlockMIDforOtherDevices;
END_GET
END_PROPERTY

PROPERTY interlockMessageWP : STRING(255)
GET
interlockMessageWP:= _interlockWPforOtherDevices;
END_GET
END_PROPERTY

PROPERTY manualMode : BOOL
GET
manualMode:= _manualMode;
END_GET
SET
_manualMode:= manualMode;
END_SET
END_PROPERTY

END_FUNCTION_BLOCK
